// Mitsubishi GX Works2 project: plc 기말 가위 바위 보 및 레이싱 카운트   PLC: Q02/Q02H

PROGRAM MAIN
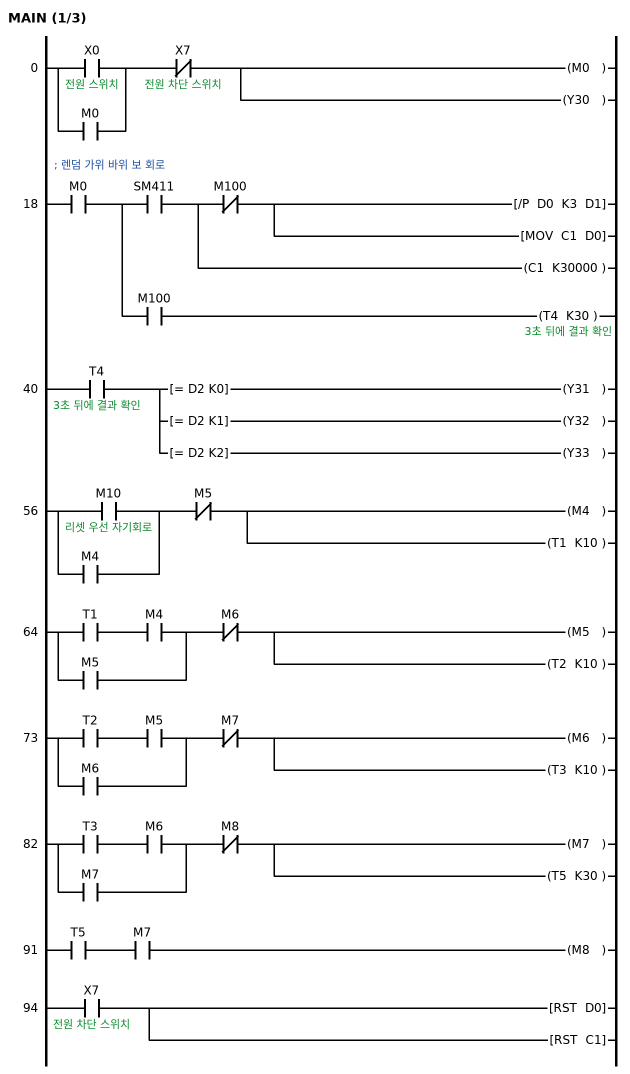
0     LD      X0  ; 전원 스위치
      OR      M0
      ANI     X7  ; 전원 차단 스위치
      OUT     M0
      OUT     Y30
; 렌덤 가위 바위 보 회로
18    LD      M0
      MPS
      AND     SM411
      MPS
      ANI     M100
      /P      D0 K3 D1
      MOV     C1 D0
      MPP
      OUT     C1 K30000
      MPP
      AND     M100
      OUT     T4 K30  ; 3초 뒤에 결과 확인
40    LD      T4  ; 3초 뒤에 결과 확인
      MPS
      AND=    D2 K0
      OUT     Y31
      MRD
      AND=    D2 K1
      OUT     Y32
      MPP
      AND=    D2 K2
      OUT     Y33
56    LD      M10  ; 리셋 우선 자기회로
      OR      M4
      ANI     M5
      OUT     M4
      OUT     T1 K10
64    LD      T1
      AND     M4
      OR      M5
      ANI     M6
      OUT     M5
      OUT     T2 K10
73    LD      T2
      AND     M5
      OR      M6
      ANI     M7
      OUT     M6
      OUT     T3 K10
82    LD      T3
      AND     M6
      OR      M7
      ANI     M8
      OUT     M7
      OUT     T5 K30
91    LD      T5
      AND     M7
      OUT     M8
94    LD      X7  ; 전원 차단 스위치
      RST     D0
      RST     C1
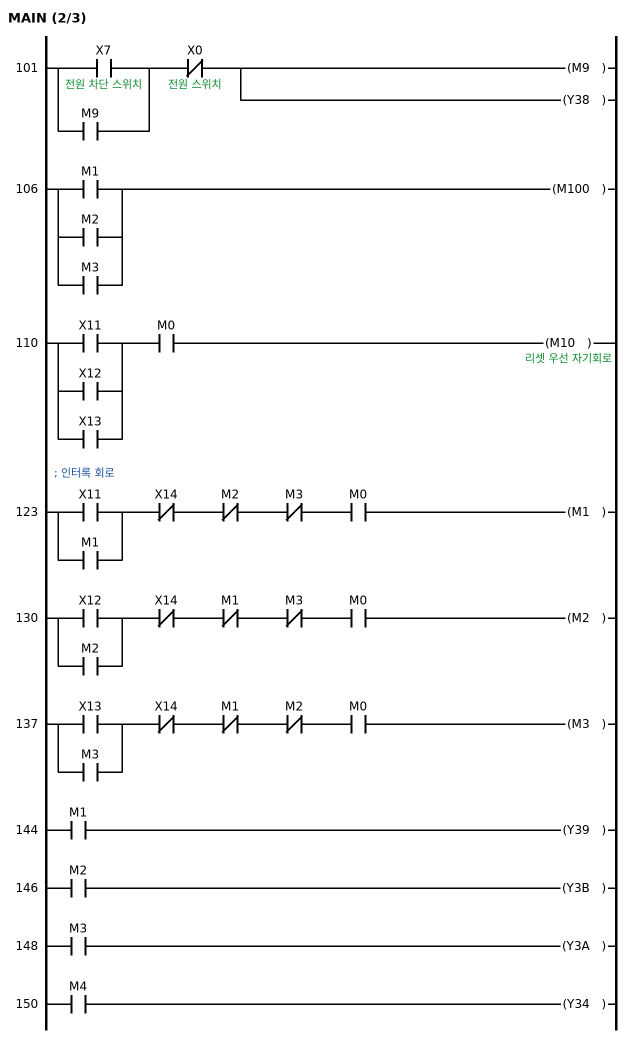
101   LD      X7  ; 전원 차단 스위치
      OR      M9
      ANI     X0  ; 전원 스위치
      OUT     M9
      OUT     Y38
106   LD      M1
      OR      M2
      OR      M3
      OUT     M100
110   LD      X11
      OR      X12
      OR      X13
      AND     M0
      OUT     M10  ; 리셋 우선 자기회로
; 인터록 회로
123   LD      X11
      OR      M1
      ANI     X14
      ANI     M2
      ANI     M3
      AND     M0
      OUT     M1
130   LD      X12
      OR      M2
      ANI     X14
      ANI     M1
      ANI     M3
      AND     M0
      OUT     M2
137   LD      X13
      OR      M3
      ANI     X14
      ANI     M1
      ANI     M2
      AND     M0
      OUT     M3
144   LD      M1
      OUT     Y39
146   LD      M2
      OUT     Y3B
148   LD      M3
      OUT     Y3A
150   LD      M4
      OUT     Y34
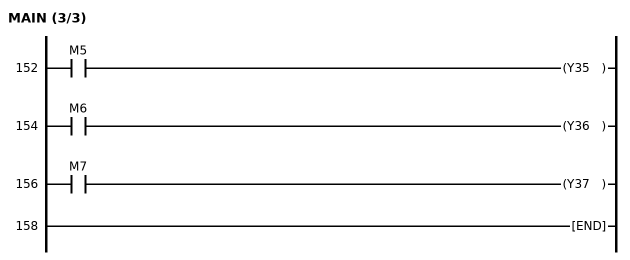
152   LD      M5
      OUT     Y35
154   LD      M6
      OUT     Y36
156   LD      M7
      OUT     Y37
158   END
END_PROGRAM
